{attribute addProperty BoxType "EK1122-0000-0018"}
{attribute addProperty Id "Beckhoff_EL5xxxsub_EK1100EK1100_179A0949162"}
{attribute addProperty CRC "4051990753"}
{attribute addProperty SizeInBites "16"}
{attribute addProperty SizeInBytes "2"}
TYPE Beckhoff_EL5xxxEK1122_F18478E1 EXTENDS EK1122_179A0949 :
STRUCT
	{attribute addProperty Name "Beckhoff_EL5xxxsub_EK1100"}
	Beckhoff_EL5xxxsub_EK1100 : EK1100_179A0949;
END_STRUCT
END_TYPE

(* stored: Version 1.2.0.0, ProductVersion 3.1.4024.9
   DUT Beckhoff_EL5xxxEK1122_F18478E1: Id {3367db89-643b-4ac1-8699-87dbc73f4ef6} *)
